(* PLC project motor1dir_1speed, Dassault Systèmes ControlBuild 2024x *)
(* stored: creationDateTime 2023-10-03T11:13:52-01:00 *)

(* This module simulates the behaviour of a motor with 1 direction and 1 speed and its electrical control logic. *)
FUNCTION_BLOCK tri_chain.motor1dir_1speed
  VAR_INPUT
    forward : BOOL := false;
    cmdSupply : BOOL := true;
    sensorSupply : BOOL := true;
    voltage380 : BOOL := true;
  END_VAR
  VAR_OUTPUT
    speedVal : REAL := 0.0;
    speedPercent : REAL := 0.0;
    thermal : BOOL := false;
    forwardFB : BOOL := false;
  END_VAR
  VAR
    increment : REAL := 0.0;
    memoFwd : BOOL := false;
    forwardState : BOOL := false;
    wantedSpeed : REAL := 0.0;
  END_VAR
  VAR CONSTANT
    nominalSpeed : REAL := 5000.0;
    nominalTime : REAL := 0.5;
    thermalLogic : BOOL := false;
    feedbackLogic : BOOL := true;
  END_VAR
  VAR
    d_locking : BOOL := false;
    v_d_locking : REAL := 0.0;
    d_feedback : BOOL := false;
    v_d_feedback : BOOL := false;
    d_electrical : BOOL := false;
    v_d_electrical : BOOL := false;
  END_VAR


ACTION C_source_code:
/* ----------------------------------------------------------------	*/
/* Type : Model of Operative Behaviour					*/
/* Category :  Associations - motors					*/
/* Author : Techniques Nouvelles d'Informatique				*/
/* Update date : October 2002						*/
/* ----------------------------------------------------------------	*/
/* This module simulates a motor with one direction and one speed	*/
/* and its electrical control logic.					*/
/* ----------------------------------------------------------------	*/


/* ----------------------------------------------------------------	*/
/* Management of orders from Control Part					*/
/*	if there is no power supply for command 				*/
/*     the contactor doesn't understand the control order		*/
/* ----------------------------------------------------------------	*/
memoFwd=forward & cmdSupply & ! d_electrical;

/* ----------------------------------------------------------------	*/
/* Calculation of the on-state of contactor				*/
/* ----------------------------------------------------------------	*/
forwardState=memoFwd & voltage380;

/* ----------------------------------------------------------------	*/
/* Management of the speed ramp						*/
/* ----------------------------------------------------------------	*/
if (d_locking) speedVal=v_d_locking;
else {
	/* Compute the increment of translation according to the simulation clock	*/
	if (nominalTime > 0.0)
		increment = (nominalSpeed/nominalTime) * (CLOCK_PERIOD/1000000.0);

	/* Compute the speed	*/
	if (forwardState) wantedSpeed = nominalSpeed;
	else wantedSpeed = 0.0;

	if ( speedVal < wantedSpeed) {
		speedVal += increment;
		if ( speedVal > wantedSpeed) speedVal = wantedSpeed;
	}
	if ( speedVal > wantedSpeed) {
		speedVal -= increment;
		if (speedVal < 0.0) speedVal = 0.0;
	}
}

/* ----------------------------------------------------------------	*/
/* Compute the percentage between the current and nominal speed	*/
/* ----------------------------------------------------------------	*/
if (nominalSpeed != 0.0)
	speedPercent = ((speedVal/nominalSpeed)*100);

/* ----------------------------------------------------------------	*/
/* Management of the thermal feedback					*/
/* ----------------------------------------------------------------	*/
if (d_electrical) thermal = v_d_electrical;
else
	if (sensorSupply) thermal = ! thermalLogic;
	else thermal = 0;


/* ----------------------------------------------------------------	*/
/* Management of feedback to Control Part					*/
/*     if a fault is required, the contactor feed-back 		*/
/*		 takes a preset state.					*/
/*	if there is no power supply for sensors 				*/
/*         contactor feed-back returns nothing				*/
/*     else contactor feed-back returns the contactor state combined	*/
/*	    with wiring logic.						*/
/* ----------------------------------------------------------------	*/
if (d_feedback) forwardFB = v_d_feedback;
else
	if (sensorSupply) forwardFB = (memoFwd ^ ! feedbackLogic);
	else forwardFB = 0;
END_ACTION
END_FUNCTION_BLOCK
